FUNCTION RestoringCWA : UINT
VAR_INPUT
	RestoreCWA : POINTER TO BOOL;
	PreviousPWA : POINTER TO UINT;
	pwa : UINT;
END_VAR
VAR
END_VAR

RestoringCWA := pwa;

IF RestoreCWA^ THEN
	RestoringCWA := PreviousPWA^;
END_IF

END_FUNCTION

(* stored: Version 1.1.0.1, ProductVersion 3.1.4024.11
   POU RestoringCWA: Id {5a22bc75-c18f-4621-9b5f-5ac2050f3afc}, SpecialFunc None *)
